PROGRAM P3_03_SP_ProcessData
VAR
	stDBParam					:ST_SPData;
	fbDBWrite					:FB_PLCDBWriteEvt(sNetId:=CONST.AMS_NETID, tTimeout:=DEFAULT_ADS_TIMEOUT);
	bWrite						:BOOL;
	tableColumns				:ARRAY [0..3] OF STRING(50) := ['Value1', 'Value2', 'Value3','DateTime'];
	arrParam					:ARRAY [0..3] OF ST_ExpParameter := [(sParaName := 'Value1', nParaSize := 101, eParaType := E_EXPPARAMETERTYPE.STRING_), 
															 (sParaName := 'Value2', nParaSize := 101, eParaType := E_EXPPARAMETERTYPE.STRING_), 
															 (sParaName := 'Value3', nParaSize := 101, eParaType := E_EXPPARAMETERTYPE.STRING_),
															 (sParaName := 'DateTime', nParaSize := 4, eParaType := E_EXPPARAMETERTYPE.DateTime)];
	fbDeleteTable    			:FB_PLCDBCmdEvt(sNetID:=CONST.AMS_NETID, tTimeout:=DEFAULT_ADS_TIMEOUT);	
	sDelete						:STRING;
	bDelete						:BOOL;
END_VAR
VAR // added by the converter: edge detectors and wires of the graphical bodies
    _rt1, _rt2 : R_TRIG;
END_VAR

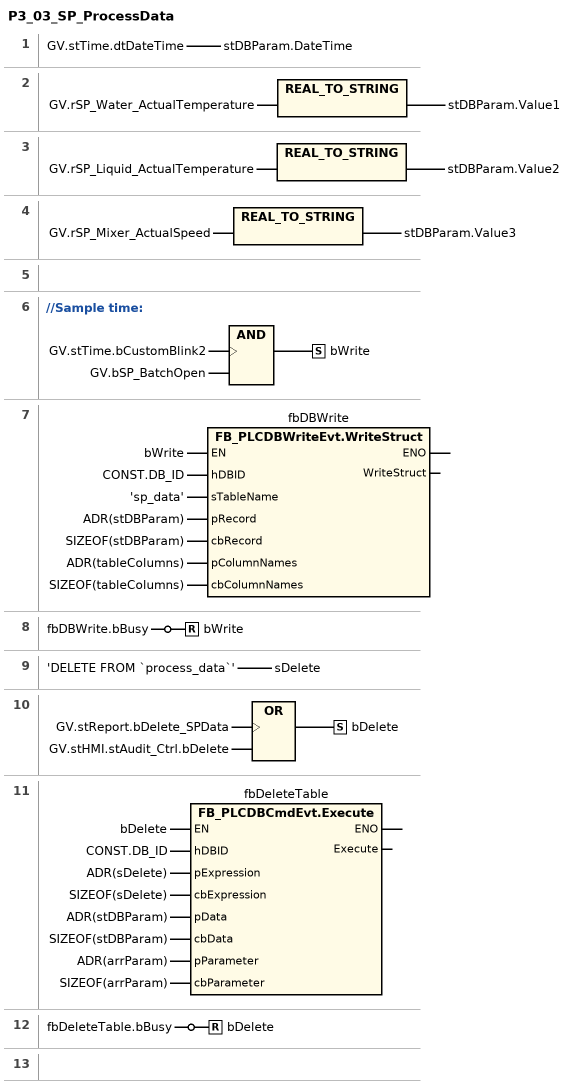
// NETWORK 1
stDBParam.DateTime := GV.stTime.dtDateTime;

// NETWORK 2
stDBParam.Value1 := REAL_TO_STRING(GV.rSP_Water_ActualTemperature);

// NETWORK 3
stDBParam.Value2 := REAL_TO_STRING(GV.rSP_Liquid_ActualTemperature);

// NETWORK 4
stDBParam.Value3 := REAL_TO_STRING(GV.rSP_Mixer_ActualSpeed);

// NETWORK 5

// NETWORK 6
// label: //Sample time
_rt1(CLK := GV.stTime.bCustomBlink2);
bWrite S= _rt1.Q AND GV.bSP_BatchOpen;

// NETWORK 7
IF bWrite THEN
    fbDBWrite.WriteStruct(
        hDBID := CONST.DB_ID,
        sTableName := 'sp_data',
        pRecord := ADR(stDBParam),
        cbRecord := SIZEOF(stDBParam),
        pColumnNames := ADR(tableColumns),
        cbColumnNames := SIZEOF(tableColumns));
END_IF

// NETWORK 8
bWrite R= NOT fbDBWrite.bBusy;

// NETWORK 9
sDelete := 'DELETE FROM `process_data`';

// NETWORK 10
_rt2(CLK := GV.stReport.bDelete_SPData);
bDelete S= _rt2.Q OR GV.stHMI.stAudit_Ctrl.bDelete;

// NETWORK 11
IF bDelete THEN
    fbDeleteTable.Execute(
        hDBID := CONST.DB_ID,
        pExpression := ADR(sDelete),
        cbExpression := SIZEOF(sDelete),
        pData := ADR(stDBParam),
        cbData := SIZEOF(stDBParam),
        pParameter := ADR(arrParam),
        cbParameter := SIZEOF(arrParam));
END_IF

// NETWORK 12
bDelete R= NOT fbDeleteTable.bBusy;

// NETWORK 13

END_PROGRAM

(* stored: Version 1.1.0.1, ProductVersion 3.1.4024.12
   POU P3_03_SP_ProcessData: Id {6160ad1b-36bc-4426-a396-a08e50144f6a}, SpecialFunc None *)
